RoboDK station: celdafin(1) (1).rdk

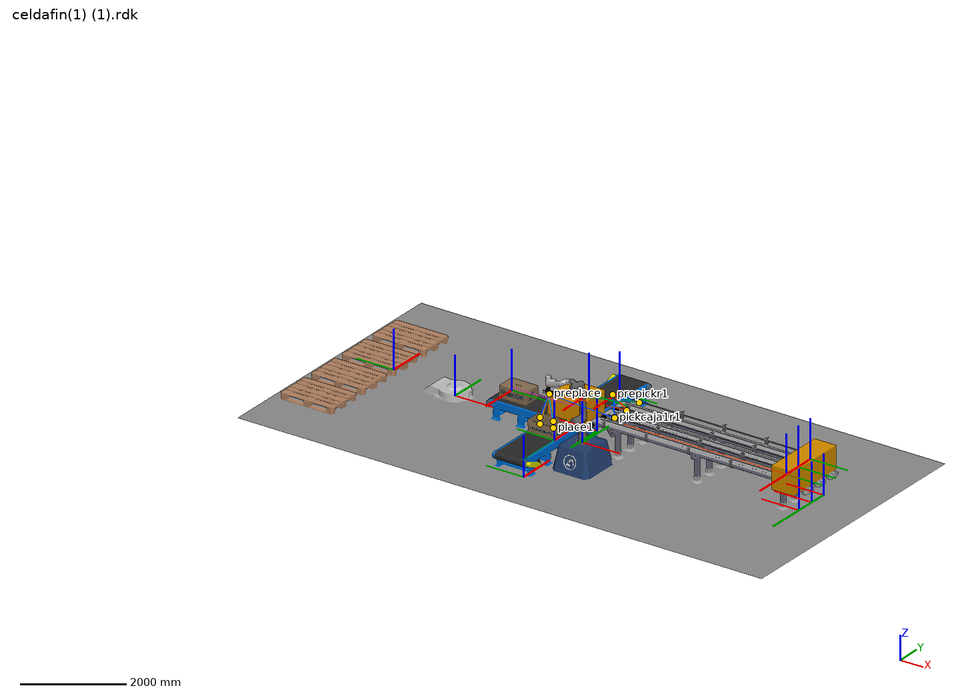
[picture v0: the station drawn from its stored meshes, robots at their saved joint values, targets as dots, program paths as lines]
Station celdafin(1) (saved by RoboDK 5.7.4). Poses are relative to the parent item; angles as X-Y-Z fixed-axis rotations.
  - folder Cintas Pequenyas
    - frame cinta1 at (4400, 800, 0) mm, rotated rx 0 ry 0 rz 180 deg
      - robot cinta1c: 1 axes
          modified DH rows (alpha deg, a mm, theta deg, d mm): 0, 0, 0, 0 linear
          base shift (0, 0, 0) mm, rotated rx 0 ry 90 rz 0 deg
          joint limits [-900000] to [900000]; home [0]; saved at [0]
        - frame caja1f at (300, 0, 0) mm, rotated rx 0 ry 0 rz 90 deg
          - object caja1 at (0, 0, 0) mm, size 199 x 305.1 x 133.7 mm, geometry from Box-12x7in-Closed.sld
          - object caja1.2 at (0, 4000, 0) mm, size 199 x 305.1 x 133.7 mm, geometry from Box-12x7in-Closed.sld
          - object caja1.3 at (0, 8000, 0) mm, size 199 x 305.1 x 133.7 mm, geometry from Box-12x7in-Closed.sld
          - object caja1.4 at (0, 12000, 0) mm, size 199 x 305.1 x 133.7 mm, geometry from Box-12x7in-Closed.sld
      - target inicinta1 (joint target) at (0, 0, 663) mm; joints [0, 0, 0, 0, 0, 0] of cinta1c
      - target fincinta1 (joint target) at (4000, 0, 663) mm; joints [4000, 0, 0, 0, 0, 0] of cinta1c
      - target fincinta1.2 (joint target) at (8000, 0, 663) mm; joints [8000, 2.845, 18.663, 0, 68.493, 170.764] of cinta1c
      - target fincinta1.3 (joint target) at (12000, 0, 663) mm; joints [12000, 2.845, 18.663, 0, 68.493, 170.764] of cinta1c
      - target fincinta1.4 (joint target) at (16000, 0, 663) mm; joints [16000, 2.845, 18.663, 0, 68.493, 170.764] of cinta1c
      - object spawn1 at (-150, -100, 500) mm, size 500 x 500 x 500 mm, geometry from Cube-500mm(1).sld
    - frame cinta2 at (4400, 1200, 0) mm, rotated rx 0 ry 0 rz 180 deg
      - robot cinta2c: 1 axes
          modified DH rows (alpha deg, a mm, theta deg, d mm): 0, 0, 0, 0 linear
          base shift (0, 0, 0) mm, rotated rx 0 ry 90 rz 0 deg
          joint limits [-900000] to [900000]; home [0]; saved at [0]
        - frame caja2f at (300, 0, 0) mm, rotated rx 0 ry 0 rz 90 deg
          - object caja2 at (0, 0, 0) mm, size 199 x 305.1 x 133.7 mm, geometry from Box-12x7in-Closed.sld
          - object caja2.2 at (0, 4000, 0) mm, size 199 x 305.1 x 133.7 mm, geometry from Box-12x7in-Closed.sld
          - object caja2.3 at (0, 8000, 0) mm, size 199 x 305.1 x 133.7 mm, geometry from Box-12x7in-Closed.sld
          - object caja2.4 at (0, 12000, 0) mm, size 199 x 305.1 x 133.7 mm, geometry from Box-12x7in-Closed.sld
      - target inicinta2 (joint target) at (0, 0, 663) mm; joints [0, 6.328, -12.115, 76.186, 22.998, -75.045] of cinta2c
      - target fincinta2 (joint target) at (4000, 0, 663) mm; joints [4000, 6.328, -12.115, 76.186, 22.998, -75.045] of cinta2c
      - target fincinta2.2 (joint target) at (8000, 0, 663) mm; joints [8000, 2.845, 18.663, 0, 68.493, 170.764] of cinta2c
      - target fincinta2.3 (joint target) at (12000, 0, 663) mm; joints [12000, 2.845, 18.663, 0, 68.493, 170.764] of cinta2c
      - target fincinta2.4 (joint target) at (16000, 0, 663) mm; joints [16000, 2.845, 18.663, 0, 68.493, 170.764] of cinta2c
      - object spawn2 at (-150, -200, 500) mm, size 500 x 500 x 500 mm, geometry from Cube-500mm(1).sld
    - frame cinta3 at (4400, 1600, 0) mm, rotated rx 0 ry 0 rz 180 deg
      - robot cinta3c: 1 axes
          modified DH rows (alpha deg, a mm, theta deg, d mm): 0, 0, 0, 0 linear
          base shift (0, 0, 0) mm, rotated rx 0 ry 90 rz 0 deg
          joint limits [-900000] to [900000]; home [0]; saved at [0]
        - frame caja3f at (300, 0, 0) mm, rotated rx 0 ry 0 rz 90 deg
          - object caja3 at (0, 0, 0) mm, size 199 x 305.1 x 133.7 mm, geometry from Box-12x7in-Closed.sld
          - object caja3.2 at (0, 4000, 0) mm, size 199 x 305.1 x 133.7 mm, geometry from Box-12x7in-Closed.sld
          - object caja3.3 at (0, 8000, 0) mm, size 199 x 305.1 x 133.7 mm, geometry from Box-12x7in-Closed.sld
          - object caja3.4 at (0, 12000, 0) mm, size 199 x 305.1 x 133.7 mm, geometry from Box-12x7in-Closed.sld
      - target inicinta3 (joint target) at (0, 0, 663) mm; joints [0, 26.9, -39.102, 77.057, 43.994, -72.284] of cinta3c
      - target fincinta3 (joint target) at (4000, 0, 663) mm; joints [4000, 26.9, -39.102, 77.057, 43.994, -72.284] of cinta3c
      - target fincinta3.2 (joint target) at (8000, 0, 663) mm; joints [8000, 2.845, 18.663, 0, 68.493, 170.764] of cinta3c
      - target fincinta3.3 (joint target) at (12000, 0, 663) mm; joints [12000, 2.845, 18.663, 0, 68.493, 170.764] of cinta3c
      - target fincinta3.4 (joint target) at (16000, 0, 663) mm; joints [16000, 2.845, 18.663, 0, 68.493, 170.764] of cinta3c
      - object spawn3 at (-150, -200, 500) mm, size 500 x 500 x 500 mm, geometry from Cube-500mm(1).sld
  - folder Cintas Grandes
    - frame cintag1 at (-650, -1000, 0) mm, rotated rx 0 ry 0 rz 90 deg
      - robot cintag1c: 1 axes
          modified DH rows (alpha deg, a mm, theta deg, d mm): 0, 0, 0, 0 linear
          base shift (0, 0, 0) mm, rotated rx 0 ry 90 rz 0 deg
          joint limits [-900000] to [900000]; home [0]; saved at [1000]
        - frame cajag1f at (0, 0, 0) mm
          - object cajag1 at (0, 0, 0) mm, size 424.8 x 637.2 x 266.3 mm, geometry from Box-24x16in-Open.sld
      - target inicintag1 (joint target) at (0, 0, 366.5) mm; joints [0, -12.476, 26.215, 0, 76.261, 75.584] of cintag1c
      - target medcintag1 (joint target) at (1000, 0, 366.5) mm; joints [1000, -12.476, 26.215, 0, 76.261, 75.584] of cintag1c
      - target fincintag1 (joint target) at (1900, 0, 366.5) mm; joints [1900, -12.476, 26.215, 0, 76.261, 75.584] of cintag1c
    - frame cintag2 at (-650, 1400, 0) mm, rotated rx 0 ry 0 rz 180 deg
      - robot cintag2c: 1 axes
          modified DH rows (alpha deg, a mm, theta deg, d mm): 0, 0, 0, 0 linear
          base shift (0, 0, 0) mm, rotated rx 0 ry 90 rz 0 deg
          joint limits [-900000] to [900000]; home [0]; saved at [1889.149]
        - frame cajag2f at (0, 100, 0) mm, rotated rx 0 ry 0 rz 90 deg
          - object cajag2 at (0, 0, 0) mm, size 398.1 x 610.2 x 267.5 mm, geometry from Box-24x16in-Closed.sld
      - object spawn4 at (-110, 200, 350) mm, size 500 x 500 x 500 mm, geometry from Cube-500mm(1).sld
      - object spawn5 at (150, 200, 350) mm, size 500 x 500 x 500 mm, geometry from Cube-500mm(1).sld
      - object spawn6 at (-110, -100, 350) mm, size 500 x 500 x 500 mm, geometry from Cube-500mm(1).sld
      - object spawn7 at (150, -100, 350) mm, size 500 x 500 x 500 mm, geometry from Cube-500mm(1).sld
      - target inicintag2 (joint target) at (520.31, 0, 366.5) mm; joints [520.306, 2.845, 18.663, 0, 68.493, 170.764] of cintag2c
      - target fincintag2 (joint target) at (1889.15, 0, 366.5) mm; joints [1889.149, 2.845, 18.663, 0, 68.493, 170.764] of cintag2c
    - frame cintag3 at (-1250, 3000, 0) mm, rotated rx 0 ry 0 rz -90 deg
      - robot cintag3c: 1 axes
          modified DH rows (alpha deg, a mm, theta deg, d mm): 0, 0, 0, 0 linear
          base shift (0, 0, 0) mm, rotated rx 0 ry 90 rz 0 deg
          joint limits [-900000] to [900000]; home [0]; saved at [1000]
        - frame cajag3f at (0, 0, 0) mm
  - folder Robots P&P
    - object pedestal at (0, 0, 0) mm, size 844.5 x 933.7 x 500 mm, geometry from Pedestal-H500mm-Type-2.sld
    - frame robot1 at (0, 0, 500) mm
      - robot robot1c (model ABB CRB 15000 10): 6 axes
          modified DH rows (alpha deg, a mm, theta deg, d mm): 0, 0, 0, 400; -90, 150, -90, 0; 0, 707, 0, 0; -90, 110, 0, 637; 90, 0, 0, 0; -90, 80, 180, 101
          joint limits [-270, -180, -225, -180, -180, -270] to [270, 180, 85, 180, 180, 270]; home [0, 0, 0, 0, 0, 0]; saved at [170.764, 2.845, 18.663, 0, 68.493, 170.764]
        - tool vacuum1, TCP at (0, 30, 180) mm, size 239 x 147 x 184.9 mm
      - target prepickr1 (Cartesian target) at (179.79, 729.43, 764.88) mm, rotated rx 180 ry 0 rz -180 deg; joints [75.584, -12.476, 26.215, 0, 76.261, 75.584] of robot1c
      - target pickcaja1r1 (Cartesian target) at (242.56, 692.28, 298.87) mm, rotated rx -180 ry 0 rz 180 deg; joints [69.885, 7.532, 55.973, 0, 26.494, 69.885] of robot1c
      - target pickcaja2r1 (Cartesian target) at (242.56, 1100, 298.87) mm, rotated rx -180 ry 0 rz -180 deg; joints [77.227, 32.053, 18.191, 0, 39.757, 77.227] of robot1c
      - target pickcaja3r1 (Cartesian target) at (242.56, 1500, 298.87) mm, rotated rx -180 ry 0 rz 180 deg; joints [80.63, 62.888, -40.371, 0, 67.483, 80.63] of robot1c
      - target preplace (Cartesian target) at (-886.42, 174.14, 693.93) mm, rotated rx -180 ry 0 rz 180 deg; joints [170.764, 2.845, 18.663, 0, 68.493, 170.764] of robot1c
      - target place1 (Cartesian target) at (-801.1, 191.84, 5.1) mm, rotated rx -180 ry 0 rz -90.88 deg; joints [166.061, 41.934, 49.678, 0, -1.613, 76.946] of robot1c
      - target place2 (Cartesian target) at (-1105.65, 196.54, 5.1) mm, rotated rx -180 ry 0 rz -90.88 deg; joints [169.669, 50.551, 19.836, 0, 19.613, 80.553] of robot1c
      - target place3 (Cartesian target) at (-801.1, 191.84, 136.05) mm, rotated rx -180 ry 0 rz -90.88 deg; joints [166.061, 28.407, 50.722, 0, 10.871, 76.945] of robot1c
      - target place4 (Cartesian target) at (-1105.65, 196.54, 135.25) mm, rotated rx -180 ry 0 rz -90.88 deg; joints [169.669, 41.597, 20.646, 0, 27.757, 80.553] of robot1c
  - folder Robots Pallets
    - frame robot3 at (-3700, 1100, 0) mm
      - robot robot3c (model ABB IRB 4400/L30 M2000): 6 axes, payload 30 kg, reach 2432 mm, repeatability 0.2 mm, weight 1040 kg
          joint limits [-165, -70, -165, -200, -120, -400] to [165, 95, 165, 200, 120, 400]; home [0, 0, 0, 0, 0, 0]; saved at [0, 0, 0, 0, 0, 0]
        - tool vacuum3, TCP at (-36, 0, 106.49) mm, size 268.4 x 184.1 x 103.7 mm
    - frame pallets at (-5100, 1100, 150) mm, rotated rx 0 ry 0 rz 90 deg
      - object pallet1 at (0, 0, 0) mm, size 800 x 1200 x 144.2 mm, geometry from Pallet-1200x800mm-Transverse(1).sld
      - object pallet2 at (1000, 0, 0) mm, size 800 x 1200 x 144.2 mm, geometry from Pallet-1200x800mm-Transverse(1).sld
      - object pallet3 at (-1000, 0, 0) mm, size 800 x 1200 x 144.2 mm, geometry from Pallet-1200x800mm-Transverse(1).sld
      - object pallet4 at (-2000, 0, 0) mm, size 800 x 1200 x 144.2 mm, geometry from Pallet-1200x800mm-Transverse(1).sld
  - folder Pisos
    - object Floor at (-2000, -500, 0) mm, size 3000 x 3000 x 0 mm, geometry from Floor(1).sld
    - object Floor1 at (1000, -500, 0) mm, size 3000 x 3000 x 0 mm, geometry from Floor(1).sld
    - object Floor2 at (4000, -500, 0) mm, size 3000 x 3000 x 0 mm, geometry from Floor(1).sld
    - object Floor3 at (4000, 2500, 0) mm, size 3000 x 3000 x 0 mm, geometry from Floor(1).sld
    - object Floor4 at (1000, 2500, 0) mm, size 3000 x 3000 x 0 mm, geometry from Floor(1).sld
    - object Floor5 at (-2000, 2500, 0) mm, size 3000 x 3000 x 0 mm, geometry from Floor(1).sld
    - object Floor6 at (-5000, 2500, 0) mm, size 3000 x 3000 x 0 mm, geometry from Floor(1).sld
    - object Floor7 at (-5000, -500, 0) mm, size 3000 x 3000 x 0 mm, geometry from Floor(1).sld
  - folder Picks
    - program p&p_caja1 (6 instructions, listed below)
    - program p&p_caja2 (6 instructions, listed below)
    - program p&p_caja3 (6 instructions, listed below)
  - folder Places
    - program place1 (5 instructions, listed below)
    - program place2 (5 instructions, listed below)
    - program place3 (5 instructions, listed below)
    - program place4 (5 instructions, listed below)
  - folder MQTT
    - Python program MqttListener (listed below)
    - Python program RobotController (listed below)
  - folder Movimiento Cinta Pequenya
    - folder CajasAUX
      - program CajasAUX1 (4 instructions, listed below)
      - program CajasAUX2 (4 instructions, listed below)
      - program CajasAUX3 (4 instructions, listed below)
    - folder MoveCinta1
      - program MoveCaja1 (4 instructions, listed below)
      - program MoveCaja1.2 (3 instructions, listed below)
      - program MoveCaja1.3 (3 instructions, listed below)
      - program MoveCaja1.4 (2 instructions, listed below)
    - folder MoveCinta2
      - program MoveCaja2 (3 instructions, listed below)
      - program MoveCaja2.2 (3 instructions, listed below)
      - program MoveCaja2.3 (3 instructions, listed below)
      - program MoveCaja2.4 (2 instructions, listed below)
    - folder MoveCinta3
      - program MoveCaja3 (3 instructions, listed below)
      - program MoveCaja3.2 (3 instructions, listed below)
      - program MoveCaja3.3 (3 instructions, listed below)
      - program MoveCaja3.4 (2 instructions, listed below)
  - folder Secuencias
    - folder 1caja
      - program 1 (3 instructions, listed below)
      - program 2 (3 instructions, listed below)
      - program 3 (3 instructions, listed below)
    - folder 2cajas
      - program 4 (6 instructions, listed below)
      - program 5 (6 instructions, listed below)
      - program 6 (6 instructions, listed below)
      - program 7 (6 instructions, listed below)
      - program 8 (6 instructions, listed below)
      - program 9 (6 instructions, listed below)
    - folder 3cajas
      - program 10 (9 instructions, listed below)
      - program 11 (9 instructions, listed below)
      - program 12 (9 instructions, listed below)
      - program 13 (9 instructions, listed below)
      - program 14 (9 instructions, listed below)
      - program 15 (9 instructions, listed below)
      - program 16 (9 instructions, listed below)
      - program 17 (9 instructions, listed below)
      - program 18 (9 instructions, listed below)
      - program 19 (9 instructions, listed below)
    - folder 4cajas
      - program 20 (12 instructions, listed below)
      - program 21 (12 instructions, listed below)
      - program 22 (12 instructions, listed below)
      - program 23 (12 instructions, listed below)
      - program 24 (12 instructions, listed below)
      - program 25 (12 instructions, listed below)
      - program 26 (12 instructions, listed below)
      - program 27 (12 instructions, listed below)
      - program 28 (12 instructions, listed below)
      - program 29 (12 instructions, listed below)
      - program 30 (12 instructions, listed below)
      - program 31 (12 instructions, listed below)
      - program 32 (12 instructions, listed below)
      - program 33 (12 instructions, listed below)
      - program 34 (12 instructions, listed below)
  - folder Paletizado
    - program Ini Caja Abierta1 (3 instructions, listed below)
    - program Fin Caja Abierta1 (2 instructions, listed below)
    - program Mov Caja Cerrada (3 instructions, listed below)
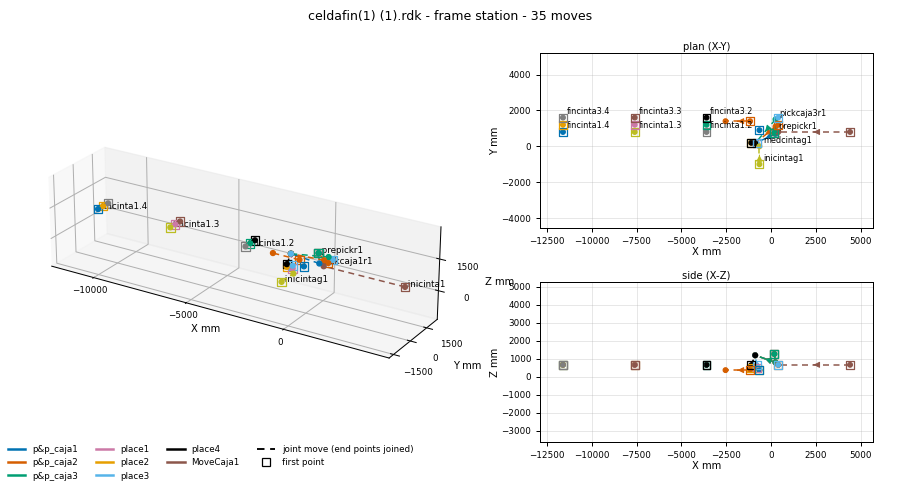
[picture p0: tool path of celdafin(1) (1).rdk in frame station, 35 of 35 moves have a stored position in this frame; points joined in program order, loops and branches not executed]

--- program p&p_caja1 (robot robot1c) ---
  Est. Ref.: robot1
  Est. herr: vacuum1
  MoveJ (prepickr1)
  MoveJ (pickcaja1r1)
  Adjuntar a vacuum1
  MoveJ (preplace)

--- program p&p_caja2 (robot robot1c) ---
  Est. Ref.: robot1
  Est. herr: vacuum1
  MoveJ (prepickr1)
  MoveJ (pickcaja2r1)
  Adjuntar a vacuum1
  MoveJ (preplace)

--- program p&p_caja3 (robot robot1c) ---
  Est. Ref.: robot1
  Est. herr: vacuum1
  MoveJ (prepickr1)
  MoveJ (pickcaja3r1)
  Adjuntar a vacuum1
  MoveJ (preplace)

--- program place1 (robot robot1c) ---
  Est. Ref.: robot1
  Est. herr: vacuum1
  MoveJ (place1)
  Separar de vacuum1
  MoveJ (preplace)

--- program place2 (robot robot1c) ---
  Est. Ref.: robot1
  Est. herr: vacuum1
  MoveJ (place2)
  Separar de vacuum1
  MoveJ (preplace)

--- program place3 (robot robot1c) ---
  Est. Ref.: robot1
  Est. herr: vacuum1
  MoveJ (place3)
  Separar de vacuum1
  MoveJ (preplace)

--- program place4 (robot robot1c) ---
  Est. Ref.: robot1
  Est. herr: vacuum1
  MoveJ (place4)
  Separar de vacuum1
  MoveJ (preplace)

--- Python program MqttListener ---
from robodk import robolink
RDK = robolink.Robolink()

import paho.mqtt.client as mqtt
import RobotController as rc

broker = "mqtt.dsic.upv.es"
port = 1883
user = "giirob"
passwd = "UPV2024"

topic_sub = "giirob/pr2/station/demo/commands"
topic_pub = "giirob/pr2/station/demo/status"


def on_message(mqttc, obj, msg):
    payload = msg.payload.decode('utf-8')
    topic = msg.topic
    qos = msg.qos
    rc.handle_message(mqttc, topic, payload)

mqttc = mqtt.Client(mqtt.CallbackAPIVersion.VERSION2)
mqttc.on_message = on_message

mqttc.username_pw_set(username=user, password=passwd)
mqttc.connect(broker, port, 60)
mqttc.subscribe(topic_sub, 0)

mqttc.publish(topic_pub, "ready 1")


mqttc.loop_forever()

--- Python program RobotController ---
from robodk import robolink
from robodk.robolink import ITEM_TYPE_PROGRAM
import threading

RDK = robolink.Robolink()

import paho.mqtt.client as mqtt

station_commands_topic = "giirob/pr2/station/demo/commands"
station_status_topic = "giirob/pr2/station/demo/status"


def handle_message(mqttc, topic, payload):
    msg = payload.strip()

    print(" Mensaje recibido:", msg)

    if topic == station_commands_topic:


        if msg == "1":
            hilo = threading.Thread(
                target=ejecutar_programa,
                args=(mqttc, "1")
            )
            hilo.start()

        elif msg == "2":
            hilo = threading.Thread(
                target=ejecutar_programa,
                args=(mqttc, "2")
            )
            hilo.start()


        elif msg == "3":
            hilo = threading.Thread(
                target=ejecutar_programa,
                args=(mqttc,"3")
            )
            hilo.start()

        elif msg == "4":
            hilo = threading.Thread(
                target=ejecutar_programa,
                args=(mqttc,"4")
            )
            hilo.start()

        elif msg == "5":
            hilo = threading.Thread(
                target=ejecutar_programa,
                args=(mqttc,"5")
            )
            hilo.start()

        elif msg == "6":
            hilo = threading.Thread(
                target=ejecutar_programa,
                args=(mqttc,"6")
            )
            hilo.start()

        elif msg == "7":
            hilo = threading.Thread(
                target=ejecutar_programa,
                args=(mqttc,"7")
            )
            hilo.start()

        elif msg == "8":
            hilo = threading.Thread(
                target=ejecutar_programa,
                args=(mqttc,"8")
            )
            hilo.start()

        elif msg == "9":
            hilo = threading.Thread(
                target=ejecutar_programa,
                args=(mqttc,"9")
            )
            hilo.start()

        elif msg == "10":
            hilo = threading.Thread(
                target=ejecutar_programa,
                args=(mqttc,"10")
            )
            hilo.start()

        elif msg == "11":
            hilo = threading.Thread(
                target=ejecutar_programa,
                args=(mqttc,"11")
            )
            hilo.start()

        elif msg == "12":
            hilo = threading.Thread(
                target=ejecutar_programa,
                args=(mqttc,"12")
            )
            hilo.start()

        elif msg == "13":
            hilo = threading.Thread(
                target=ejecutar_programa,
                args=(mqttc,"13")
            )
            hilo.start()

        elif msg == "14":
            hilo = threading.Thread(
                target=ejecutar_programa,
                args=(mqttc,"14")
            )
            hilo.start()

        elif msg == "15":
            hilo = threading.Thread(
                target=ejecutar_programa,
                args=(mqttc,"15")
            )
            hilo.start()

        elif msg == "16":
            hilo = threading.Thread(
                target=ejecutar_programa,
                args=(mqttc,"16")
            )
            hilo.start()

        elif msg == "17":
            hilo = threading.Thread(
                target=ejecutar_programa,
                args=(mqttc,"17")
            )
            hilo.start()

        elif msg == "18":
            hilo = threading.Thread(
                target=ejecutar_programa,
                args=(mqttc,"18")
            )
            hilo.start()

        elif msg == "19":
            hilo = threading.Thread(
                target=ejecutar_programa,
                args=(mqttc,"19")
            )
            hilo.start()

        elif msg == "20":
            hilo = threading.Thread(
                target=ejecutar_programa,
                args=(mqttc,"20")
            )
            hilo.start()

        elif msg == "21":
            hilo = threading.Thread(
                target=ejecutar_programa,
                args=(mqttc,"21")
            )
            hilo.start()

        elif msg == "22":
            hilo = threading.Thread(
                target=ejecutar_programa,
                args=(mqttc,"22")
            )
            hilo.start()

        elif msg == "23":
            hilo = threading.Thread(
                target=ejecutar_programa,
                args=(mqttc,"23")
            )
            hilo.start()

        elif msg == "24":
            hilo = threading.Thread(
                target=ejecutar_programa,
                args=(mqttc,"24")
            )
            hilo.start()

        elif msg == "25":
            hilo = threading.Thread(
                target=ejecutar_programa,
                args=(mqttc,"25")
            )
            hilo.start()

        elif msg == "26":
            hilo = threading.Thread(
                target=ejecutar_programa,
                args=(mqttc,"26")
            )
            hilo.start()

        elif msg == "27":
            hilo = threading.Thread(
                target=ejecutar_programa,
                args=(mqttc,"27")
            )
            hilo.start()

        elif msg == "28":
            hilo = threading.Thread(
                target=ejecutar_programa,
                args=(mqttc,"28")
            )
            hilo.start()

        elif msg == "29":
            hilo = threading.Thread(
                target=ejecutar_programa,
                args=(mqttc,"29")
            )
            hilo.start()

        elif msg == "30":
            hilo = threading.Thread(
                target=ejecutar_programa,
                args=(mqttc,"30")
            )
            hilo.start()

        elif msg == "31":
            hilo = threading.Thread(
                target=ejecutar_programa,
                args=(mqttc,"31")
            )
            hilo.start()

        elif msg == "32":
            hilo = threading.Thread(
                target=ejecutar_programa,
                args=(mqttc,"32")
            )
            hilo.start()

        elif msg == "33":
            hilo = threading.Thread(
                target=ejecutar_programa,
                args=(mqttc,"33")
            )
            hilo.start()

        elif msg == "34":
            hilo = threading.Thread(
                target=ejecutar_programa,
                args=(mqttc,"34")
            )
            hilo.start()





         # else:
            #print("Comando no reconocido")


def ejecutar_programa(mqttc, nombre_programa):
    programa = RDK.Item(nombre_programa, ITEM_TYPE_PROGRAM)
    programa.RunProgram()

--- program CajasAUX1 (robot robot1c) ---
  Est. Ref.: cinta1
  Ocultar caja1.2
  Ocultar caja1.3
  Ocultar caja1.4

--- program CajasAUX2 (robot robot1c) ---
  Est. Ref.: cinta2
  Ocultar caja2.2
  Ocultar caja2.3
  Ocultar caja2.4

--- program CajasAUX3 (robot robot1c) ---
  Est. Ref.: cinta3
  Ocultar caja3.2
  Ocultar caja3.3
  Ocultar caja3.4

--- program MoveCaja1 (robot cinta1c) ---
  Est. Ref.: cinta1
  MoveJ (inicinta1)
  MoveJ (fincinta1)
  Mostrar caja1.2

--- program MoveCaja1.2 (robot cinta1c) ---
  Est. Ref.: cinta1
  MoveJ (fincinta1.2)
  Mostrar caja1.3

--- program MoveCaja1.3 (robot cinta1c) ---
  Est. Ref.: cinta1
  MoveJ (fincinta1.3)
  Mostrar caja1.4

--- program MoveCaja1.4 (robot cinta1c) ---
  Est. Ref.: cinta1
  MoveJ (fincinta1.4)

--- program MoveCaja2 (robot cinta2c) ---
  Est. Ref.: cinta2
  MoveJ (fincinta2)
  Mostrar caja2.2

--- program MoveCaja2.2 (robot cinta2c) ---
  Est. Ref.: cinta2
  MoveJ (fincinta2.2)
  Mostrar caja2.3

--- program MoveCaja2.3 (robot cinta2c) ---
  Est. Ref.: cinta2
  MoveJ (fincinta2.3)
  Mostrar caja2.4

--- program MoveCaja2.4 (robot cinta2c) ---
  Est. Ref.: cinta2
  MoveJ (fincinta2.4)

--- program MoveCaja3 (robot cinta3c) ---
  Est. Ref.: cinta3
  MoveJ (fincinta3)
  Mostrar caja3.2

--- program MoveCaja3.2 (robot cinta3c) ---
  Est. Ref.: cinta3
  MoveJ (fincinta3.2)
  Mostrar caja3.3

--- program MoveCaja3.3 (robot cinta3c) ---
  Est. Ref.: cinta3
  MoveJ (fincinta3.3)
  Mostrar caja3.4

--- program MoveCaja3.4 (robot cinta3c) ---
  Est. Ref.: cinta3
  MoveJ (fincinta3.4)

--- program 1 (robot robot1c) ---
  Llamar MoveCaja1
  Llamar p&p_caja1
  Llamar place1

--- program 2 (robot robot1c) ---
  Llamar MoveCaja2
  Llamar p&p_caja2
  Llamar place1

--- program 3 (robot robot1c) ---
  Llamar MoveCaja3
  Llamar p&p_caja3
  Llamar place1

--- program 4 (robot cinta1c) ---
  Llamar MoveCaja1
  Llamar p&p_caja1
  Llamar place1
  Llamar MoveCaja1.2
  Llamar p&p_caja1
  Llamar place2

--- program 5 (robot cinta1c) ---
  Llamar MoveCaja1
  Llamar p&p_caja1
  Llamar place1
  Llamar MoveCaja2
  Llamar p&p_caja2
  Llamar place2

--- program 6 (robot cinta1c) ---
  Llamar MoveCaja1
  Llamar p&p_caja1
  Llamar place1
  Llamar MoveCaja3
  Llamar p&p_caja3
  Llamar place2

--- program 7 (robot cinta1c) ---
  Llamar MoveCaja2
  Llamar p&p_caja2
  Llamar place1
  Llamar MoveCaja2.2
  Llamar p&p_caja2
  Llamar place2

--- program 8 (robot cinta1c) ---
  Llamar MoveCaja2
  Llamar p&p_caja2
  Llamar place1
  Llamar MoveCaja3
  Llamar p&p_caja3
  Llamar place2

--- program 9 (robot cinta1c) ---
  Llamar MoveCaja3
  Llamar p&p_caja3
  Llamar place1
  Llamar MoveCaja3.2
  Llamar p&p_caja3
  Llamar place2

--- program 10 (robot cinta1c) ---
  Llamar MoveCaja1
  Llamar p&p_caja1
  Llamar place1
  Llamar MoveCaja1.2
  Llamar p&p_caja1
  Llamar place2
  Llamar MoveCaja1.3
  Llamar p&p_caja1
  Llamar place3

--- program 11 (robot cinta1c) ---
  Llamar MoveCaja1
  Llamar p&p_caja1
  Llamar place1
  Llamar MoveCaja1.2
  Llamar p&p_caja1
  Llamar place2
  Llamar MoveCaja2
  Llamar p&p_caja2
  Llamar place3

--- program 12 (robot cinta1c) ---
  Llamar MoveCaja1
  Llamar p&p_caja1
  Llamar place1
  Llamar MoveCaja1.2
  Llamar p&p_caja1
  Llamar place2
  Llamar MoveCaja3
  Llamar p&p_caja3
  Llamar place3

--- program 13 (robot cinta1c) ---
  Llamar MoveCaja1
  Llamar p&p_caja1
  Llamar place1
  Llamar MoveCaja2
  Llamar p&p_caja2
  Llamar place2
  Llamar MoveCaja2.2
  Llamar p&p_caja2
  Llamar place3

--- program 14 (robot cinta1c) ---
  Llamar MoveCaja1
  Llamar p&p_caja1
  Llamar place1
  Llamar MoveCaja2
  Llamar p&p_caja2
  Llamar place2
  Llamar MoveCaja3
  Llamar p&p_caja3
  Llamar place3

--- program 15 (robot cinta1c) ---
  Llamar MoveCaja1
  Llamar p&p_caja1
  Llamar place1
  Llamar MoveCaja2
  Llamar p&p_caja2
  Llamar place2
  Llamar MoveCaja2.2
  Llamar p&p_caja2
  Llamar place3

--- program 16 (robot cinta1c) ---
  Llamar MoveCaja2
  Llamar p&p_caja2
  Llamar place1
  Llamar MoveCaja2.2
  Llamar p&p_caja2
  Llamar place2
  Llamar MoveCaja2.3
  Llamar p&p_caja2
  Llamar place3

--- program 17 (robot cinta1c) ---
  Llamar MoveCaja2
  Llamar p&p_caja2
  Llamar place1
  Llamar MoveCaja2.2
  Llamar p&p_caja2
  Llamar place2
  Llamar MoveCaja3
  Llamar p&p_caja3
  Llamar place3

--- program 18 (robot cinta1c) ---
  Llamar MoveCaja2
  Llamar p&p_caja2
  Llamar place1
  Llamar MoveCaja3
  Llamar p&p_caja3
  Llamar place2
  Llamar MoveCaja3.2
  Llamar p&p_caja3
  Llamar place3

--- program 19 (robot cinta1c) ---
  Llamar MoveCaja3
  Llamar p&p_caja3
  Llamar place1
  Llamar MoveCaja3.2
  Llamar p&p_caja3
  Llamar place2
  Llamar MoveCaja3.3
  Llamar p&p_caja3
  Llamar place3

--- program 20 (robot cinta1c) ---
  Llamar MoveCaja1
  Llamar p&p_caja1
  Llamar place1
  Llamar MoveCaja1.2
  Llamar p&p_caja1
  Llamar place2
  Llamar MoveCaja1.3
  Llamar p&p_caja1
  Llamar place3
  Llamar MoveCaja1.4
  Llamar p&p_caja1
  Llamar place4

--- program 21 (robot cinta1c) ---
  Llamar MoveCaja1
  Llamar p&p_caja1
  Llamar place1
  Llamar MoveCaja1.2
  Llamar p&p_caja1
  Llamar place2
  Llamar MoveCaja1.3
  Llamar p&p_caja1
  Llamar place3
  Llamar MoveCaja2
  Llamar p&p_caja2
  Llamar place4

--- program 22 (robot cinta1c) ---
  Llamar MoveCaja1
  Llamar p&p_caja1
  Llamar place1
  Llamar MoveCaja1.2
  Llamar p&p_caja1
  Llamar place2
  Llamar MoveCaja1.3
  Llamar p&p_caja1
  Llamar place3
  Llamar MoveCaja3
  Llamar p&p_caja3
  Llamar place4

--- program 23 (robot cinta1c) ---
  Llamar MoveCaja1
  Llamar p&p_caja1
  Llamar place1
  Llamar MoveCaja1.2
  Llamar p&p_caja1
  Llamar place2
  Llamar MoveCaja2
  Llamar p&p_caja2
  Llamar place3
  Llamar MoveCaja2.2
  Llamar p&p_caja2
  Llamar place4

--- program 24 (robot cinta1c) ---
  Llamar MoveCaja1
  Llamar p&p_caja1
  Llamar place1
  Llamar MoveCaja1.2
  Llamar p&p_caja1
  Llamar place2
  Llamar MoveCaja2
  Llamar p&p_caja2
  Llamar place3
  Llamar MoveCaja3
  Llamar p&p_caja3
  Llamar place4

--- program 25 (robot cinta1c) ---
  Llamar MoveCaja1
  Llamar p&p_caja1
  Llamar place1
  Llamar MoveCaja1.2
  Llamar p&p_caja1
  Llamar place2
  Llamar MoveCaja3
  Llamar p&p_caja3
  Llamar place3
  Llamar MoveCaja3.2
  Llamar p&p_caja3
  Llamar place4

--- program 26 (robot cinta1c) ---
  Llamar MoveCaja1
  Llamar p&p_caja1
  Llamar place1
  Llamar MoveCaja2
  Llamar p&p_caja2
  Llamar place2
  Llamar MoveCaja2.2
  Llamar p&p_caja2
  Llamar place3
  Llamar MoveCaja2.3
  Llamar p&p_caja2
  Llamar place4

--- program 27 (robot cinta1c) ---
  Llamar MoveCaja1
  Llamar p&p_caja1
  Llamar place1
  Llamar MoveCaja2
  Llamar p&p_caja2
  Llamar place2
  Llamar MoveCaja2.2
  Llamar p&p_caja2
  Llamar place3
  Llamar MoveCaja3
  Llamar p&p_caja3
  Llamar place4

--- program 28 (robot cinta1c) ---
  Llamar MoveCaja1
  Llamar p&p_caja1
  Llamar place1
  Llamar MoveCaja2
  Llamar p&p_caja2
  Llamar place2
  Llamar MoveCaja3
  Llamar p&p_caja3
  Llamar place3
  Llamar MoveCaja3.2
  Llamar p&p_caja3
  Llamar place4

--- program 29 (robot cinta1c) ---
  Llamar MoveCaja1
  Llamar p&p_caja1
  Llamar place1
  Llamar MoveCaja3
  Llamar p&p_caja3
  Llamar place2
  Llamar MoveCaja3.2
  Llamar p&p_caja3
  Llamar place3
  Llamar MoveCaja3.3
  Llamar p&p_caja3
  Llamar place4

--- program 30 (robot cinta1c) ---
  Llamar MoveCaja2
  Llamar p&p_caja2
  Llamar place1
  Llamar MoveCaja2.2
  Llamar p&p_caja2
  Llamar place2
  Llamar MoveCaja2.3
  Llamar p&p_caja2
  Llamar place3
  Llamar MoveCaja2.4
  Llamar p&p_caja2
  Llamar place4

--- program 31 (robot cinta1c) ---
  Llamar MoveCaja2
  Llamar p&p_caja2
  Llamar place1
  Llamar MoveCaja2.2
  Llamar p&p_caja2
  Llamar place2
  Llamar MoveCaja2.3
  Llamar p&p_caja2
  Llamar place3
  Llamar MoveCaja3
  Llamar p&p_caja3
  Llamar place4

--- program 32 (robot cinta1c) ---
  Llamar MoveCaja2
  Llamar p&p_caja2
  Llamar place1
  Llamar MoveCaja2.2
  Llamar p&p_caja2
  Llamar place2
  Llamar MoveCaja3
  Llamar p&p_caja3
  Llamar place3
  Llamar MoveCaja3.2
  Llamar p&p_caja3
  Llamar place4

--- program 33 (robot cinta1c) ---
  Llamar MoveCaja2
  Llamar p&p_caja2
  Llamar place1
  Llamar MoveCaja3
  Llamar p&p_caja3
  Llamar place2
  Llamar MoveCaja3.2
  Llamar p&p_caja3
  Llamar place3
  Llamar MoveCaja3.3
  Llamar p&p_caja3
  Llamar place4

--- program 34 (robot cinta1c) ---
  Llamar MoveCaja3
  Llamar p&p_caja3
  Llamar place1
  Llamar MoveCaja3.2
  Llamar p&p_caja3
  Llamar place2
  Llamar MoveCaja3.3
  Llamar p&p_caja3
  Llamar place3
  Llamar MoveCaja3.4
  Llamar p&p_caja3
  Llamar place4

--- program Ini Caja Abierta1 (robot cintag1c) ---
  Est. Ref.: cintag1
  MoveJ (inicintag1)
  MoveJ (medcintag1)

--- program Fin Caja Abierta1 (robot cintag1c) ---
  Est. Ref.: cintag1
  MoveJ (fincintag1)

--- program Mov Caja Cerrada (robot cintag2c) ---
  Est. Ref.: cintag2
  MoveJ (inicintag2)
  MoveJ (fincintag2)
